FUNCTION_BLOCK FB_Bel_Input
VAR_INPUT
	IN_Leistung					: BYTE;
	IN_Dali_Arc_Error			: BOOL;
	IN_Dali_Off_Error			: BOOL;
	IN_Dali_Error				: BOOL;
END_VAR
VAR_OUTPUT
	Leistung					: BYTE;
	Stoerung					: BOOL;
END_VAR
VAR
END_VAR

Leistung					:=REAL_TO_BYTE((IN_Leistung-126)/1.28);
Stoerung					:=IN_Dali_Arc_Error OR IN_Dali_Arc_Error OR IN_Dali_Error;

END_FUNCTION_BLOCK

(* stored: Version 1.1.0.1, ProductVersion 3.1.4024.9
   POU FB_Bel_Input: Id {5022a524-2b4f-41e4-9900-bffef008928c}, SpecialFunc None *)
